// TIA Portal V19 export
FUNCTION "A03_HMI_CALL" : Void   // FC227, LAD
// stored: SetENOAutomatically false
BEGIN

REGION Network 1
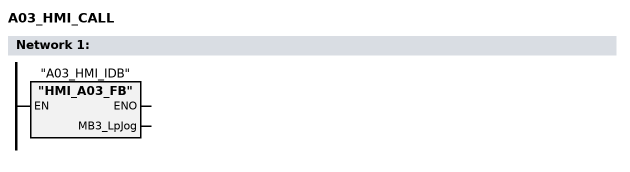
   RUNG wire#powerrail
      "A03_HMI_IDB"(MB3_LpJog =>)
   END_RUNG
   // the same network as SCL:
   "A03_HMI_IDB"();   // "HMI_A03_FB"
END_REGION
END_FUNCTION
